// Mitsubishi GX Works2 project: biogas   PLC: FX3U/FX3UC

PROGRAM MAIN
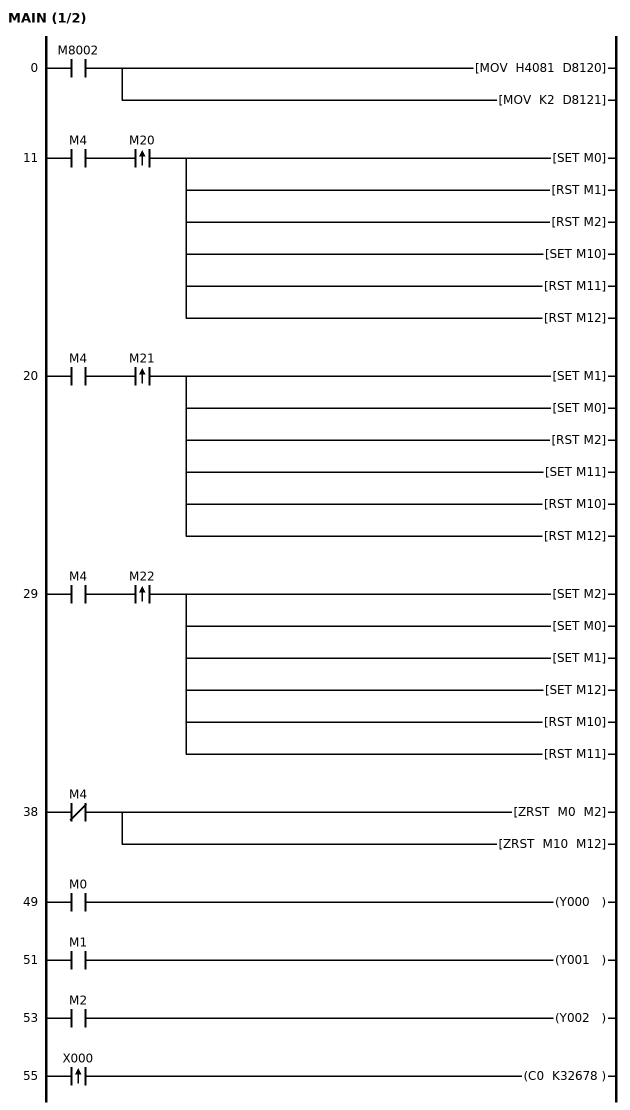
0     LD      M8002
      MOV     H4081 D8120
      MOV     K2 D8121
11    LD      M4
      ANDP    M20
      SET     M0
      RST     M1
      RST     M2
      SET     M10
      RST     M11
      RST     M12
20    LD      M4
      ANDP    M21
      SET     M1
      SET     M0
      RST     M2
      SET     M11
      RST     M10
      RST     M12
29    LD      M4
      ANDP    M22
      SET     M2
      SET     M0
      SET     M1
      SET     M12
      RST     M10
      RST     M11
38    LDI     M4
      ZRST    M0 M2
      ZRST    M10 M12
49    LD      M0
      OUT     Y000
51    LD      M1
      OUT     Y001
53    LD      M2
      OUT     Y002
55    LDP     X000
      OUT     C0 K32678
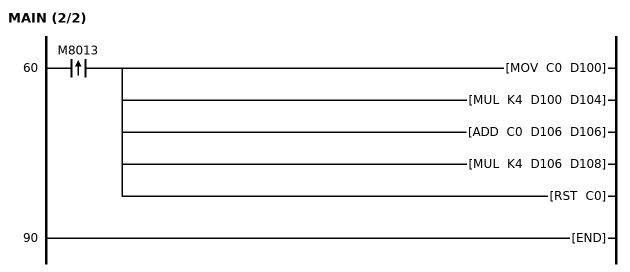
60    LDP     M8013
      MOV     C0 D100
      MUL     K4 D100 D104
      ADD     C0 D106 D106
      MUL     K4 D106 D108
      RST     C0
90    END
END_PROGRAM
